FUNCTION_BLOCK IO_force
VAR_INPUT
	Raw_IO : BOOL;
END_VAR

VAR_OUTPUT
	Out : BOOL;
END_VAR

VAR
	ForceEnable : BOOL;
	ForceStatus : BOOL;
END_VAR

IF NOT ForceEnable THEN
	OUT := Raw_IO;
ELSE
	OUT := ForceStatus;
END_IF

END_FUNCTION_BLOCK

(* stored: Version 1.1.0.1, ProductVersion 3.1.4024.14
   POU IO_force: Id {9f2c4e8d-5cf0-44e7-85f0-68ef135972a0}, SpecialFunc None *)
